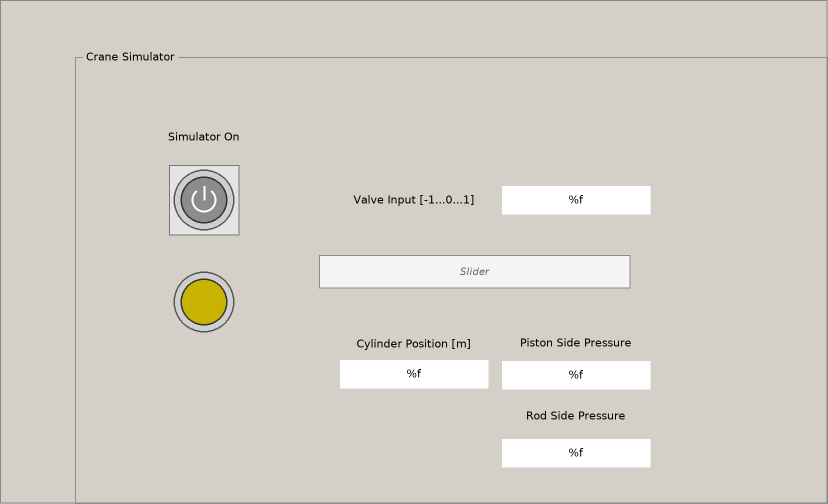
VISUALIZATION Visualization  // 828x504
    GroupBox (75,49 753x455), "Crane Simulator"
        Lamp1 (94,218 70x70), variable: P_CraneSim.bSimulatorOn, style: Lamp-Lamp1-Yellow
        PowerSwitch (94,116 70x70), variable: P_CraneSim.bSimulatorOn, behaviour: TOGGLE, style: Switch-PowerSwitch-Gray
        Slider (244,206 311x33), variable: P_CraneSim.fValeInput, scale -1..1
        Textfield (426,311 150x30), "%f", text variable: P_CraneSim.fPistonSidePressure
        Textfield (264,310 150x30), "%f", text variable: P_CraneSim.fCylinderPosition
        Textfield (426,389 150x30), "%f", text variable: P_CraneSim.fRodSidePressure
        Textfield (426,136 150x30), "%f", text variable: P_CraneSim.fValeInput
        Label (54,73 150x30), "Simulator On"
        Label (426,279 150x30), "Piston Side Pressure"
        Label (426,352 150x30), "Rod Side Pressure"
        Label (264,136 150x30), "Valve Input [-1...0...1]"
        Label (264,280 150x30), "Cylinder Position [m]"
END_VISUALIZATION

(* stored: Version 1.1.0.1, ProductVersion 3.1.4024.12
   Visu Visualization: Id {2d1790f2-dc71-4492-8f4a-0451002747e8} *)
